INTERFACE I_PushButton

PROPERTY PUBLIC isPressed : BOOL
GET
END_GET
END_PROPERTY

PROPERTY PUBLIC isReleased : BOOL
GET
END_GET
END_PROPERTY

END_INTERFACE

(* stored: Version 1.1.0.1, ProductVersion 3.1.4024.12
   Itf I_PushButton: Id {fe549dec-5ff8-47ac-9537-a7beef6b3b28}
   Property isPressed: Id {b920ace0-d2c4-473f-9e37-262e83d49d1a}
   Get Get: Id {0069a615-c887-45f8-a4ac-44510ec6387e}
   Property isReleased: Id {9bc13ae3-a644-4b24-8f14-23bf6f9c7b64}
   Get Get: Id {88b40e50-d4b0-42c4-a9f2-a73f4db36ac5} *)
